# EPICS autosave request: support/areaDetector-s55/iocBoot/iocMAR345/auto_settings.req
file "ADBase_settings.req",       P=$(P),  R=cam1:
file "mar345_settings.req",       P=$(P),  R=cam1:
file "NDFile_settings.req",       P=$(P),  R=cam1:
file "commonPlugin_settings.req", P=$(P)
